TYPE "Positioning_MOL_Machine_Par"
VERSION : 0.1
// Block: Positioning_MOL_Machine_Par
   STRUCT
      PosTolerance : LReal;
      DelayInPosition : Time;
      Minus_Limit : LReal;
      Plus_Limit : LReal;
      PreCutOff : LReal;
   END_STRUCT;

END_TYPE
